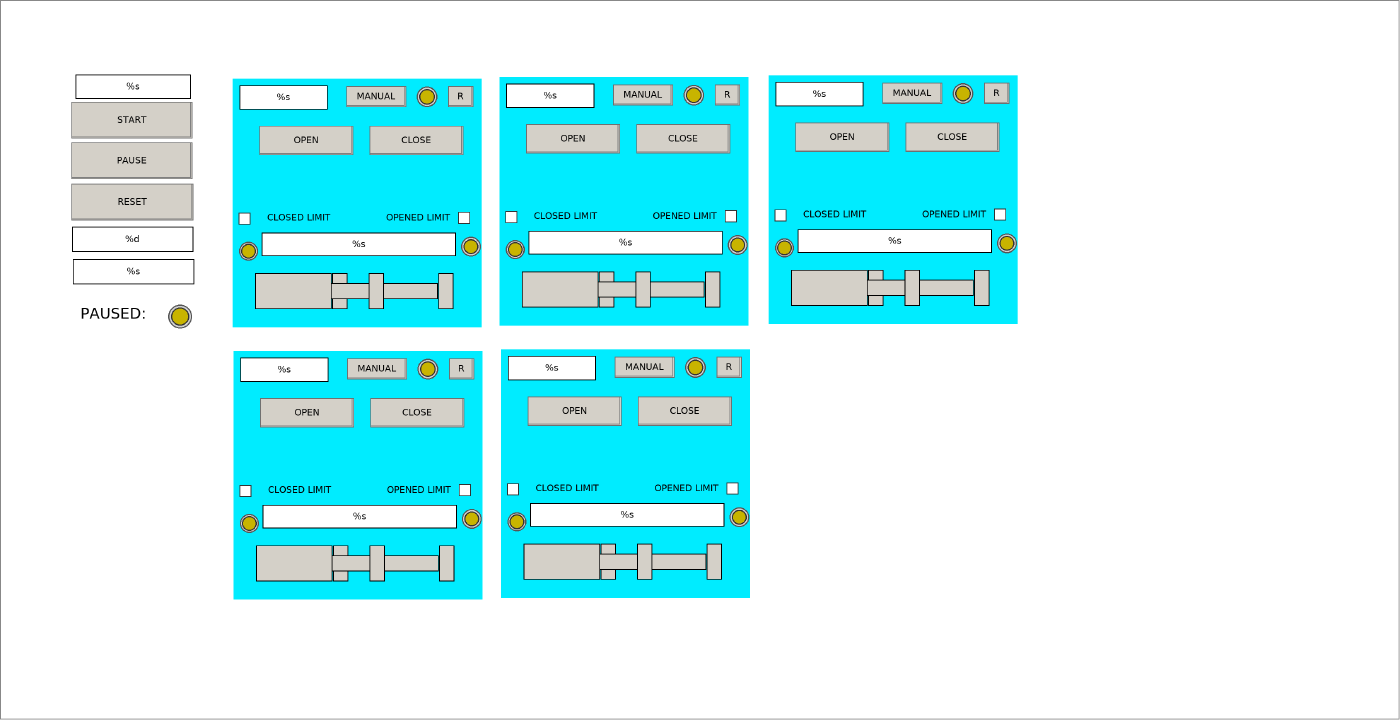
VISUALIZATION vFEEDER  // 1690x870
VAR_IN_OUT
	vFEEDER: FB_FEEDER;
END_VAR
    Frame (281,95 300x300)
        shows vPISTON(PIST1 := vFEEDER.fbPUSH)
    Frame (603,93 300x300)
        shows vPISTON(PIST1 := vFEEDER.fbHOLD1)
    Frame (928,91 300x300)
        shows vPISTON(PIST1 := vFEEDER.fbHOLD2)
    Frame (67,89 200x360)
        shows vSTATION_CONTROLLER(vSTATION := vFEEDER)
    Frame (282,424 300x300)
        shows vPISTON(PIST1 := vFEEDER.fbOPEN1)
    Frame (605,422 300x300)
        shows vPISTON(PIST1 := vFEEDER.fbOPEN1)
END_VISUALIZATION

// ---- POUs/STATIONS/vSEPARATE.TcVIS
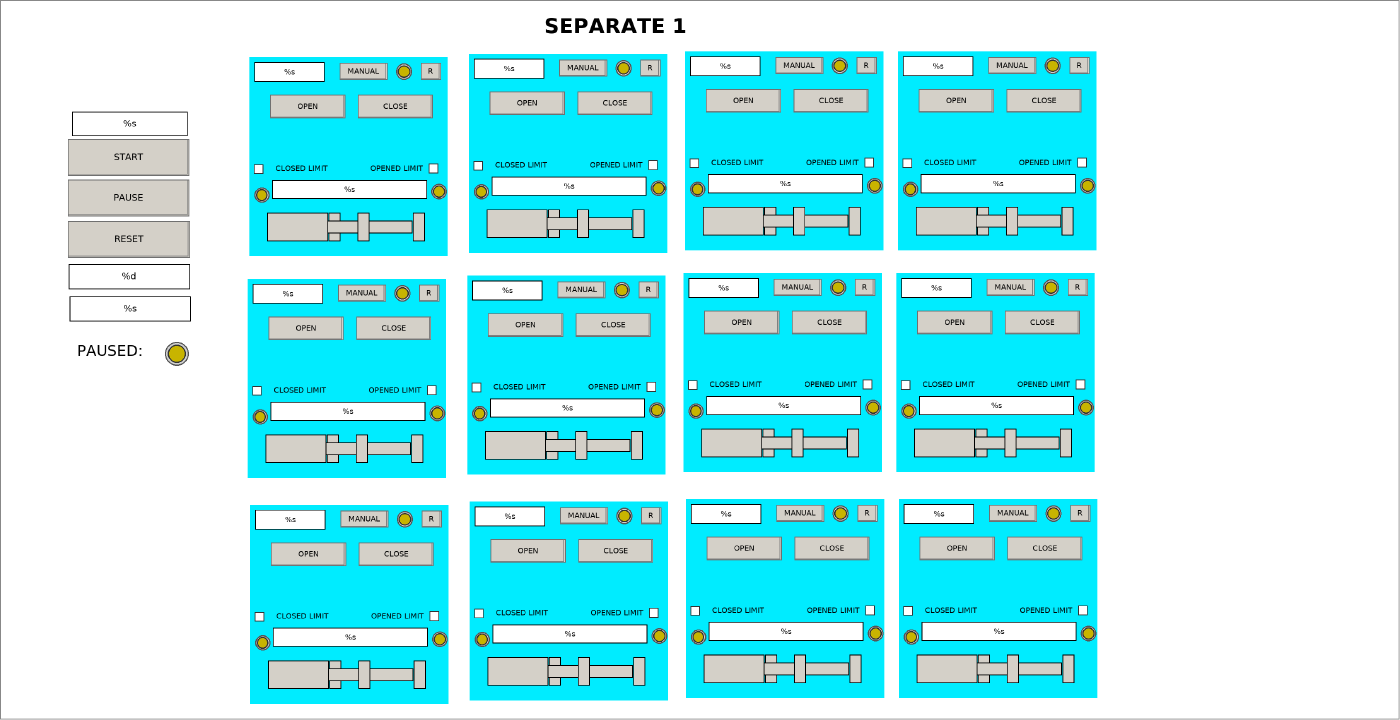
VISUALIZATION vSEPARATE  // 1690x870
VAR_IN_OUT
	vSEPARATE: FB_SEPARATE;
END_VAR
    Frame (301,69 239x240)
        shows vPISTON(PIST1 := vSEPARATE1.fbPIST1)
    Frame (63,134 200x360)
        shows vSTATION_CONTROLLER(vSTATION := vSEPARATE1)
    Label (605,16 276x30), "SEPARATE 1"
    Frame (566,65 239x240)
        shows vPISTON(PIST1 := vSEPARATE1.fbPIST1)
    Frame (827,62 239x240)
        shows vPISTON(PIST1 := vSEPARATE1.fbPIST1)
    Frame (1084,62 239x240)
        shows vPISTON(PIST1 := vSEPARATE1.fbPIST1)
    Frame (299,337 239x240)
        shows vPISTON(PIST1 := vSEPARATE1.fbPIST1)
    Frame (564,333 239x240)
        shows vPISTON(PIST1 := vSEPARATE1.fbPIST1)
    Frame (825,330 239x240)
        shows vPISTON(PIST1 := vSEPARATE1.fbPIST1)
    Frame (1082,330 239x240)
        shows vPISTON(PIST1 := vSEPARATE1.fbPIST1)
    Frame (302,610 239x240)
        shows vPISTON(PIST1 := vSEPARATE1.fbPIST1)
    Frame (567,606 239x240)
        shows vPISTON(PIST1 := vSEPARATE1.fbPIST1)
    Frame (828,603 239x240)
        shows vPISTON(PIST1 := vSEPARATE1.fbPIST1)
    Frame (1085,603 239x240)
        shows vPISTON(PIST1 := vSEPARATE1.fbPIST1)
END_VISUALIZATION

// ---- POUs/STATIONS/vSTATION_CONTROLLER.TcVIS
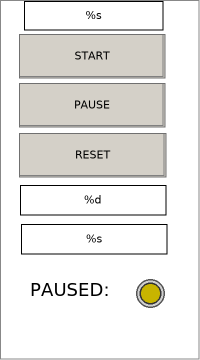
VISUALIZATION vSTATION_CONTROLLER  // 200x360
VAR_IN_OUT
	vSTATION : FB_STATION;
END_VAR
    Button (19,34 146x44), "START"
        OnMouseClick: execute { vSTATION.aSTART(); }
    Button (19,133 147x44), "RESET"
        OnMouseClick: execute { vSTATION.bRESET:=TRUE; }
    Rectangle (20,185 146x30), "%d", text variable: vSTATION.iSTATION_STATE
    Rectangle (21,224 146x30), "%s", text variable: vSTATION.sSTATION_STATE
    Button (19,83 146x44), "PAUSE"
        toggle vSTATION.bPAUSE
    Lamp1 (134,272 33x43), variable: vSTATION.bPAUSE, style: Lamp-Lamp1-Yellow
    Label (26,275 88x30), "PAUSED:"
    Rectangle (24,1 139x29), "%s", text variable: vSTATION.sName
END_VISUALIZATION

// ---- VISUs/vCOMM.TcVIS
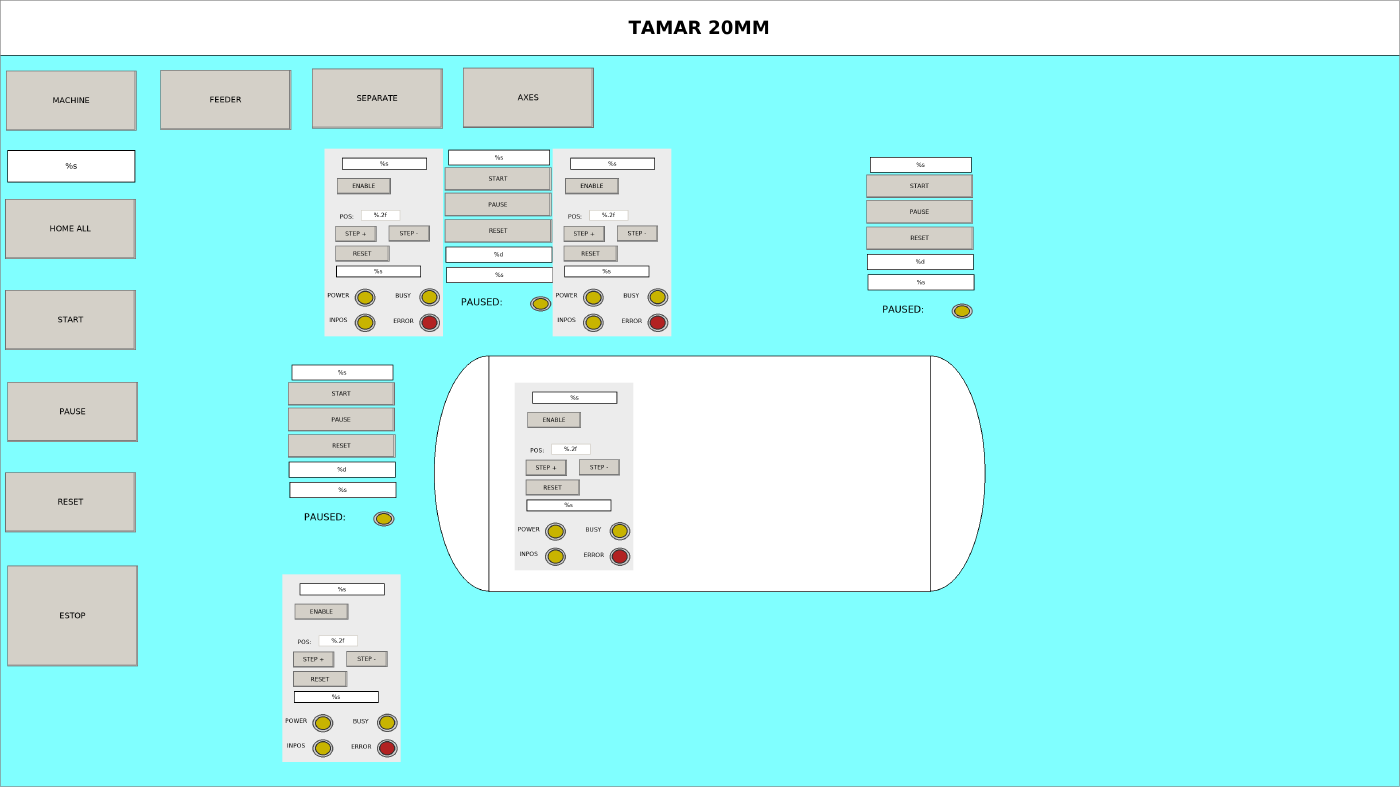
VISUALIZATION vCOMM  // 1920x1080
    Button (7,398 179x82), "START", input disabled if: NOT bMAIN_HOMED
        OnMouseClick: execute { bMAIN_START:=TRUE; }
    Rectangle (-3,-1 1924x77), "TAMAR 20MM"
    Button (10,524 179x82), "PAUSE"
    Button (7,648 179x82), "RESET"
        OnMouseClick: execute { bMAIN_RESET:=TRUE; }
    Button (10,776 179x138), "ESTOP"
    Frame (266,199 1690x870)
        shows vMACHINE()
        shows vFEEDER(vFEEDER := fbFEEDER)
        shows vSEPARATE(vSEPARATE := fbSEPARATE1)
        shows AXES_SCREEN()
    Button (220,96 179x82), "FEEDER"
        OnMouseClick: FrameSelectionChange Selection=SelectedFrame=00e59953-e4a5-4fe1-b8af-e2191fac8d98, Selection=1, GlobSel=AssignType=Directly, SelType=Locally
    Button (8,97 179x82), "MACHINE"
        OnMouseClick: FrameSelectionChange Selection=SelectedFrame=00e59953-e4a5-4fe1-b8af-e2191fac8d98, GlobSel=AssignType=Directly, SelType=Locally
    Button (428,94 179x82), "SEPARATE"
        OnMouseClick: FrameSelectionChange Selection=SelectedFrame=00e59953-e4a5-4fe1-b8af-e2191fac8d98, Selection=2, GlobSel=AssignType=Directly, SelType=Locally
    Rectangle (10,206 175x44), "%s", text variable: sMAIN_STATE
    Button (635,93 179x82), "AXES"
        OnMouseClick: FrameSelectionChange Selection=SelectedFrame=00e59953-e4a5-4fe1-b8af-e2191fac8d98, Selection=3, GlobSel=AssignType=Directly, SelType=Locally
    Button (7,273 179x82), "HOME ALL"
        OnMouseClick: execute { bMAIN_HOME:=TRUE; }
END_VISUALIZATION

// ---- VISUs/vMACHINE.TcVIS
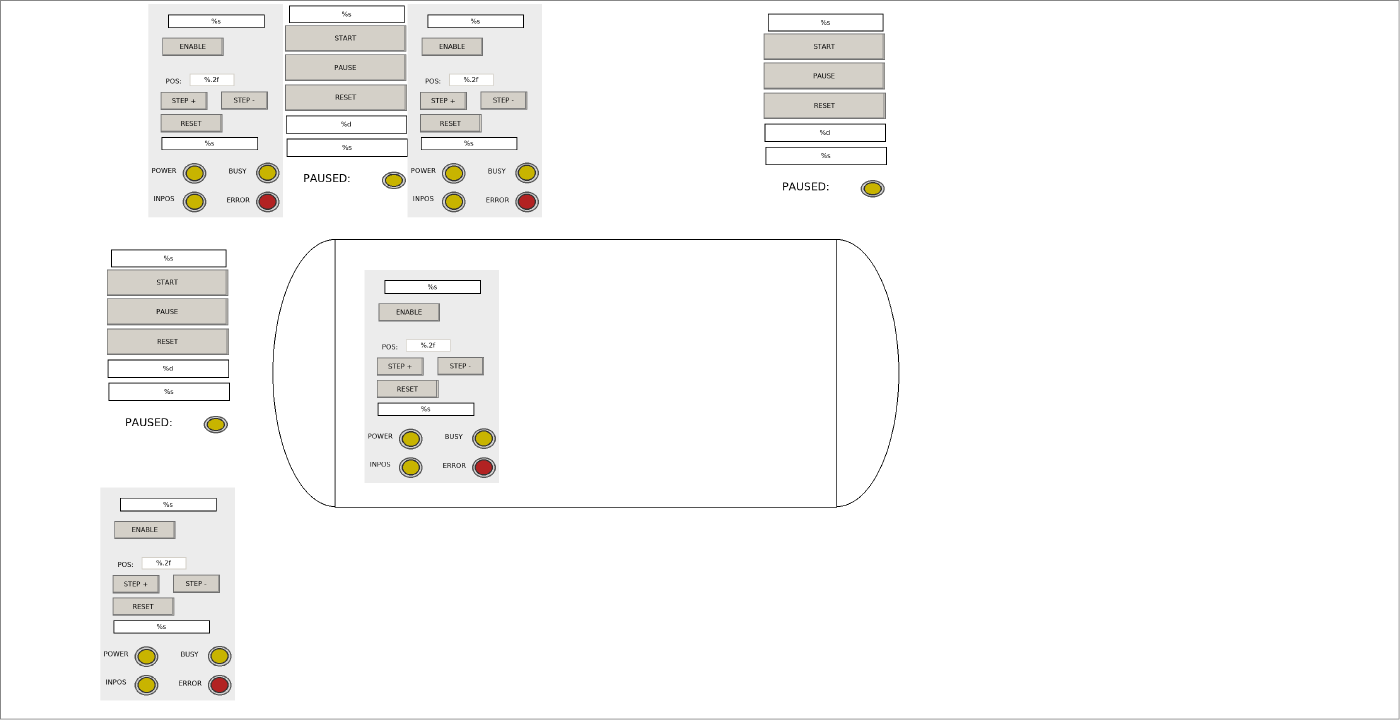
VISUALIZATION vMACHINE  // 1690x870
    Frame (110,301 200x260)
        shows vSTATION_CONTROLLER(vSTATION := fbFEEDER)
    Frame (325,6 200x260)
        shows vSTATION_CONTROLLER(vSTATION := fbSEPARATE1)
    Frame (903,16 200x260)
        shows vSTATION_CONTROLLER(vSTATION := fbSEPARATE2)
    Ellipse (329,289 150x323)
    Ellipse (935,289 150x323)
    Rectangle (404,289 606x324)
    Frame (440,326 162x257)
        shows vAXIS_CONTROLLER(vAXIS := MAIN_CONV)
    Frame (121,589 162x257)
        shows vAXIS_CONTROLLER(vAXIS := SUP_CONV)
    Frame (492,5 162x257)
        shows vAXIS_CONTROLLER(vAXIS := PRESS1B)
    Frame (179,5 162x257)
        shows vAXIS_CONTROLLER(vAXIS := PRESS1A)
END_VISUALIZATION
